PROGRAM MAIN
VAR
	// trigger command execution for OpenWeatherMap samples 	
	bGetOpenWeatherMap 				: BOOL; 

	fbHttpClientOpenWeatherMap		: FB_IotHttpClient :=(sHostName:='api.openweathermap.org',
								  	bKeepAlive:=TRUE,	tConnectionTimeout:=T#10S);

	fbHttpGetOpenWeatherMap			: FB_TestHTTP_Get_openWeatherMap;
END_VAR

// init client parameters at startup
IF NOT fbHttpClientOpenWeatherMap.bConfigured THEN 
	fbHttpClientOpenWeatherMap.nHostPort:= 443;
	fbHttpClientOpenWeatherMap.stTLS.bNoServerCertCheck:= TRUE;
END_IF

IF fbHttpClientOpenWeatherMap.bConfigured THEN
 	fbHttpGetOpenWeatherMap(bSend:=bGetOpenWeatherMap, fbClient:=fbHttpClientOpenWeatherMap);
END_IF

fbHttpClientOpenWeatherMap.Execute();

END_PROGRAM

(* stored: Version 1.1.0.1, ProductVersion 3.1.4024.6
   POU MAIN: Id {df8ef25c-63ca-48ff-b97a-e5f69f6c7e3e}, SpecialFunc None *)
